INTERFACE I_CommandAbortingState

METHOD PUBLIC SetAborted
VAR_INPUT
END_VAR
END_METHOD

METHOD PUBLIC SetError
VAR_INPUT
	ErrorId : UDINT;
END_VAR
END_METHOD

END_INTERFACE

(* stored: Version 1.1.0.1, ProductVersion 3.1.4024.12
   Itf I_CommandAbortingState: Id {98b6f948-2305-4709-8b4a-ea1e3a13afd2}
   Method SetAborted: Id {30339df6-20c9-4d2f-bee6-5f41d46d7353}
   Method SetError: Id {642271fb-4115-4982-80d4-f8d76a7b6e1c} *)
